// SIMATIC S7-200 project (STEP 7-Micro/WIN), CPU 214 REL 01.11

SYMBOL_TABLE ANWENDER1
S7_enable        V12.7    // Slave 7 Enable-Flag
ASi_Input_Reg_D  VD0      // Input Register
Opt_NS           V0.7     // optischer Näherungsschalter
Kap_NS           V0.6     // kapazitiver Näherungsschalter
Ein_LS           V0.4     // Ein Lichtschranke
Tast_3           V0.3     // Taster 3
Tast_2           V0.2     // Taster 2
Tast_1           V0.1     // Taster 1
Tast_0           V0.0     // Taster 0
MagE_U           V1.6     // magnetischer Endschalter oben
MagE_D           V1.5     // magnetischer Endschalter unten
Glas_LS          V1.4     // Glas Lichtschranke
ZEnd_Up          V1.1     // Endschalter Zylinder oben
ZEnd_Do          V1.0     // Endschalter Zylinder unten
IndNS_2          V2.6     // induktiver Näherungsschalter Bit2
IndNS_1          V2.5     // induktiver Näherungsschalter Bit1
IndNS_0          V2.4     // induktiver Näherungsschalter Bit0
Sonar_2          V2.2     // Sonar Bit2
Sonar_1          V2.1     // Sonar Bit1
Sonar_0          V2.0     // Sonar Bit0
Pressure         VW4      // Zylinderdruck
Distance         VW6      // Distanz
Joy_X            VW8      // Joystick X-Achse
Joy_Y            VW10     // Joystick Y-Achse
ASi_OutputReg_D  VD12     // Output Register
S2_enable        V12.2    // Slave 2 Enable-Flag
S3_enable        V12.3    // Slave 3 Enable-Flag
S5_enable        V12.5    // Slave 5 Enable-Flag
MC_Dir           V15.7    // Motorcontroller Direction
MC_Go            V15.6    // Motorcontroller Go
Zyl_Up           V15.5    // Zylinder Auf
Zyl_Do           V15.4    // Zylinder Ab
Lampe_3          V15.3    // Lampe 3
Lampe_2          V15.2    // Lampe 2
Lampe_1          V15.1    // Lampe 1
Lampe_0          V15.0    // Lampe 0
DVM              VW16     // Digital Voltmeter
MCSpeed          VW18     // Motorspeed
END_SYMBOL_TABLE

SYMBOL_TABLE DP
CP_Con           I2.4     // Blockkonsitenter Datentransfer
CP_Ready         I2.1     // CP 242-8 Ready
CP_Com           Q2.5     // Auftragsbit (Softwarehandshake)
CP_Res           I2.5     // Antwortbit (Softwarehandshake)
END_SYMBOL_TABLE

ORGANIZATION_BLOCK MAIN:OB1
TITLE=Demoprogramm zur Verwendung der ASi-Lib (Dieter Etz)
// 
BEGIN
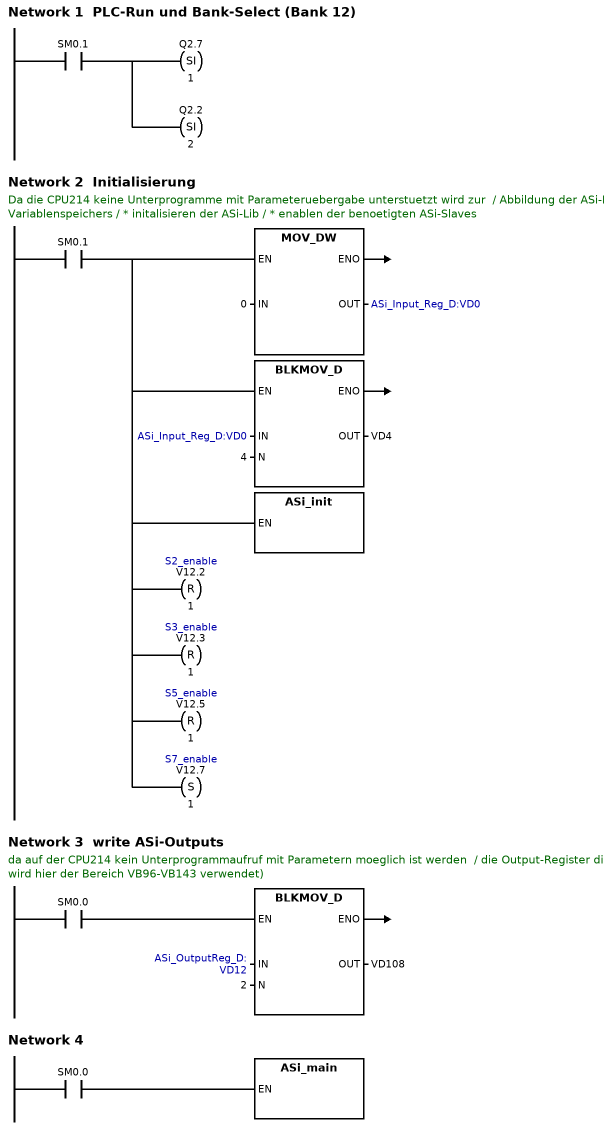
Network 1 // PLC-Run und Bank-Select (Bank 12)
// 
// 
LD     SM0.1
SI     Q2.7, 1
SI     Q2.2, 2
Network 2 // Initialisierung
// Da die CPU214 keine Unterprogramme mit Parameteruebergabe unterstuetzt wird zur 
// Abbildung der ASi-Komponenten der Variablenspeicher VD0 - VD16 verwendet.
// * loeschen des verwendeten Variablenspeichers
// * initalisieren der ASi-Lib
// * enablen der benoetigten ASi-Slaves
LD     SM0.1
MOVD   0, ASi_Input_Reg_D:VD0
BMD    ASi_Input_Reg_D:VD0, VD4, 4
CALL   ASi_init:SBR1
R      S2_enable:V12.2, 1
R      S3_enable:V12.3, 1
R      S5_enable:V12.5, 1
S      S7_enable:V12.7, 1
Network 3 // write ASi-Outputs
// da auf der CPU214 kein Unterprogrammaufruf mit Parametern moeglich ist werden 
// die Output-Register direkt in den Speicherbereich der Library kopiert
// (als Speicherbereich fuer die Bibliothek wird hier der Bereich VB96-VB143 verwendet)
LD     SM0.0
BMD    ASi_OutputReg_D:VD12, VD108, 2
Network 4
LD     SM0.0
CALL   ASi_main:SBR3
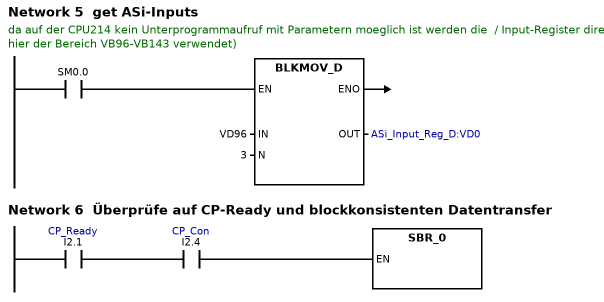
Network 5 // get ASi-Inputs
// da auf der CPU214 kein Unterprogrammaufruf mit Parametern moeglich ist werden die 
// Input-Register direkt vom Speicherbereich der Library kopiert
// (als Speicherbereich fuer die Bibliothek wird hier der Bereich VB96-VB143 verwendet)
LD     SM0.0
BMD    VD96, ASi_Input_Reg_D:VD0, 3
Network 6 // Überprüfe auf CP-Ready und blockkonsistenten Datentransfer
// 
// 
LD     CP_Ready:I2.1
A      CP_Con:I2.4
CALL   SBR_0:SBR0
END_ORGANIZATION_BLOCK

SUBROUTINE_BLOCK SBR_0:SBR0
TITLE=UNTERPROGRAMM-KOMMENTARE
BEGIN
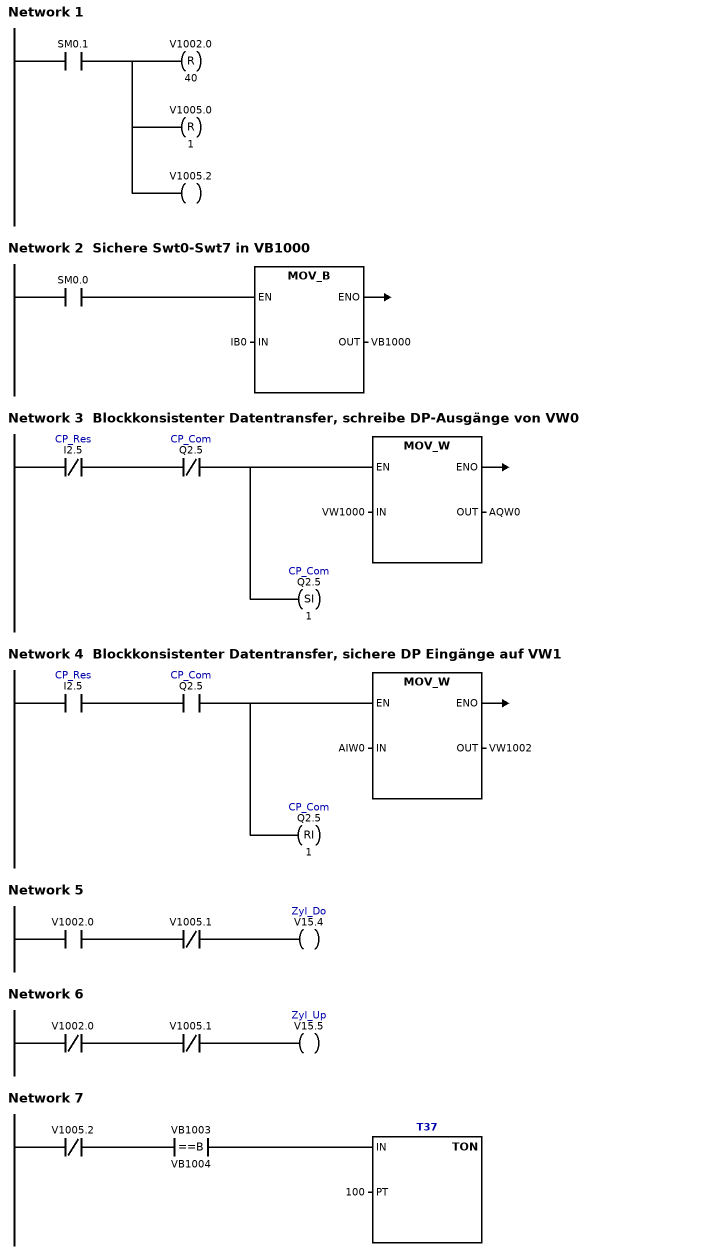
Network 1
LD     SM0.1
R      V1002.0, 40
R      V1005.0, 1
=      V1005.2
Network 2 // Sichere Swt0-Swt7 in VB1000
LD     SM0.0
MOVB   IB0, VB1000
Network 3 // Blockkonsistenter Datentransfer, schreibe DP-Ausgänge von VW0
LDN    CP_Res:I2.5
AN     CP_Com:Q2.5
MOVW   VW1000, AQW0
SI     CP_Com:Q2.5, 1
Network 4 // Blockkonsistenter Datentransfer, sichere DP Eingänge auf VW1
LD     CP_Res:I2.5
A      CP_Com:Q2.5
MOVW   AIW0, VW1002
RI     CP_Com:Q2.5, 1
Network 5
LD     V1002.0
AN     V1005.1
=      Zyl_Do:V15.4
Network 6
LDN    V1002.0
AN     V1005.1
=      Zyl_Up:V15.5
Network 7
LDN    V1005.2
AB=    VB1003, VB1004
TON    T37, 100
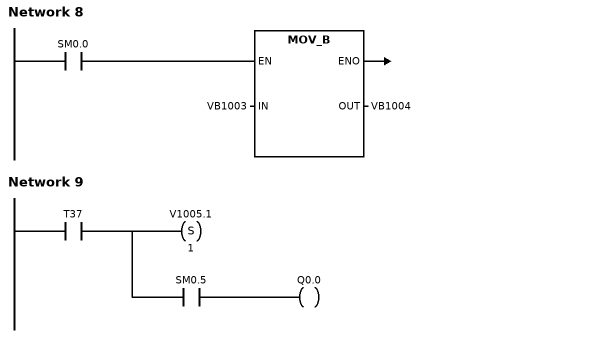
Network 8
LD     SM0.0
MOVB   VB1003, VB1004
Network 9
LD     T37
S      V1005.1, 1
A      SM0.5
=      Q0.0
END_SUBROUTINE_BLOCK

// SBR1: protected block, not included

// SBR2: protected block, not included

// SBR3: protected block, not included

// SBR4: protected block, not included

// SBR5: protected block, not included
